FUNCTION_BLOCK ExtendUnwrap IMPLEMENTS I_Unwrapper
VAR
	_x : UDINT;
	_y : UDINT;
END_VAR

METHOD Sample : BOOL
VAR_INPUT
	ImageWidth	: UDINT;
	ImageHeight	: UDINT;
	XOffset	: UDINT;
	YOffset	: UDINT;
END_VAR
_x	   := MIN(ImageWidth - 1, XOffset);
_y	   := MIN(ImageHeight - 1, YOffset);
Sample := TRUE;
END_METHOD

PROPERTY X : UDINT
GET
X := _x;
END_GET
END_PROPERTY

PROPERTY Y : UDINT
GET
Y := _y;
END_GET
END_PROPERTY

END_FUNCTION_BLOCK

(* stored: Version 1.1.0.1
   POU ExtendUnwrap: Id {bc3707c6-fcc6-4bc8-b2b0-6de6b06d61b1}, SpecialFunc None
   Method Sample: Id {ba9870d3-46bf-4503-9de3-59e5319e4f41}
   Property X: Id {72ce8925-d899-4f57-9f09-783a873a6368}
   Get Get: Id {bf15af2b-59bb-4ede-be82-28c68b757c66}
   Property Y: Id {3907860d-61ae-4620-8887-bc6893eb3b89}
   Get Get: Id {5fcd8691-7577-4513-8984-4aa1f1408b21} *)
